// Implicitly generated code : DO NOT EDIT
FUNCTION CheckBounds : DINT
VAR_INPUT
    index, lower, upper : DINT;
END_VAR
// User defined local variables
VAR
    sMessageLow : STRING := 'CheckBounds: Index too low (%d)';
    sMessageHigh : STRING := 'CheckBounds: Index too high (%d)';
END_VAR

// Implicitly generated code : Only an Implementation suggestion
{noflow}
IF index < lower THEN
    CheckBounds := lower;
    ADSLOGDINT(msgCtrlMask := ADSLOG_MSGTYPE_ERROR, msgFmtStr := sMessageLow, dintArg := index);
ELSIF index > upper THEN
    CheckBounds := upper;
    ADSLOGDINT(msgCtrlMask := ADSLOG_MSGTYPE_ERROR, msgFmtStr := sMessageHigh, dintArg := index);
ELSE
    CheckBounds := index;
END_IF

{flow}

END_FUNCTION

(* stored: Version 1.1.0.1
   POU CheckBounds: Id {c12686d1-6980-00bb-27af-81d22ca6d6a2}, SpecialFunc CheckBounds *)
